Staubli VAL3: onSave.pgx

public program onSave(string& x_sItem[])
  local num i
  local num l_nSize
  local num l_nIndex
begin
  //if bToSave
  // update
  if isDefined(pt:tTraj[pEditPoint.sID])
    // to prevent error on the executing update the nIndex
    pEditPoint.nIndex=pt:tTraj[pEditPoint.sID].nIndex
    // copy the value
    pt:tTraj[pEditPoint.sID]=pEditPoint
    // link the frame
    call pt:link_all(pEditPoint.sID)
  endIf
  // saveIt
  pt:libSave()
  bToSave=false
  //endIf
end
